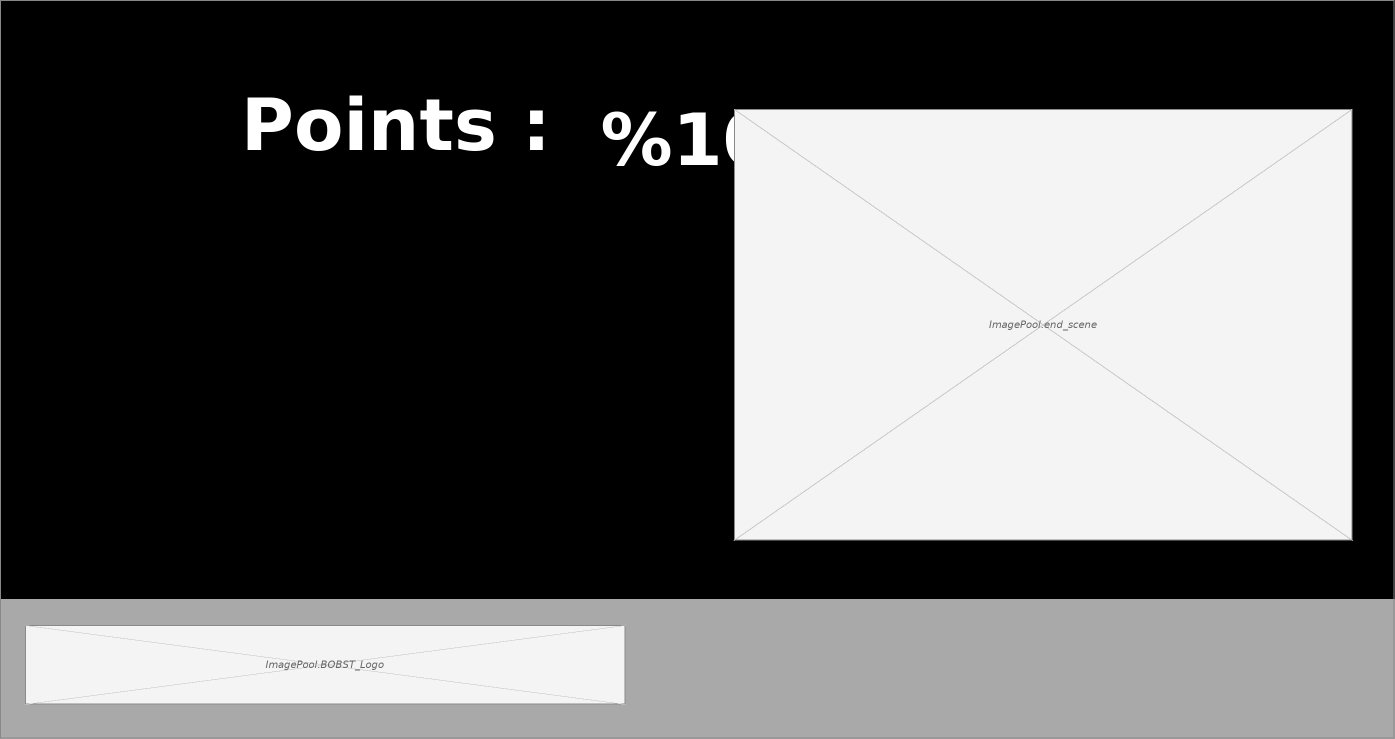
VISUALIZATION V_Fin_Match  // 1395x739
    Rectangle (0,599 1396x140)
    Textfield (516,75 450x129), "%10.0f", text variable: G_Match.PointMatch
    Textfield (158,60 476x129), "Points :"
    Image (25,625 600x79), image: ImagePool.BOBST_Logo
        OnMouseDown: change screen: V_Menu
    Image (734,109 618x431), image: ImagePool.end_scene
END_VISUALIZATION

(* stored: Version 1.1.0.1, ProductVersion 3.1.4024.12
   Visu V_Fin_Match: Id {be37c65a-99c2-4549-b090-7b3a665d4724} *)
